{attribute 'linkalways'} 
{attribute 'no_explicit_call' := 'This FB is a CLASS and must be accessed using methods or properties'}
{attribute 'enable_dynamic_creation'}
FUNCTION_BLOCK Node_F_VN_ConvertCartesianToPolarPoints EXTENDS VisionNode
VAR
	ipSrcPointsCart : _ITcVnContainer;
    ipDestPointsPolar : _ITcVnContainer;
    hrPrev : _HRESULT(S_OK);
	hresult : _HRESULT(S_OK);
END_VAR

METHOD PUBLIC  Clone : I_Node
VAR
	pNode : POINTER TO Node_F_VN_ConvertCartesianToPolarPoints;
END_VAR
pNode := __NEW(Node_F_VN_ConvertCartesianToPolarPoints);
Clone := pNode^;
END_METHOD

METHOD FB_init : BOOL
VAR_INPUT
	bInitRetains : BOOL; // if TRUE, the retain variables are initialized (warm start / cold start)
	bInCopyCode : BOOL;  // if TRUE, the instance afterwards gets moved into the copy code (online change)
END_VAR
AddInput('ipSrcPointsCart', ipSrcPointsCart);
AddInput('hrPrev', hrPrev);
AddOutput('ipDestPointsPolar', ipDestPointsPolar);
AddOutput('hresult',hresult);
END_METHOD

METHOD PROTECTED OnExecute
hresult.Value := F_VN_ConvertCartesianToPolarPoints(
	ipSrcPointsCart := ipSrcPointsCart.Value,
	ipDestPointsPolar := ipDestPointsPolar.Value,
	hrPrev := hrPrev.Value);
END_METHOD

METHOD PUBLIC PreExecutionCheck
VAR_INPUT
	Check : I_PreExecutionChecks;
END_VAR
Check.IsTrue(ipSrcPointsCart.IsValid, 'ipSrcPointsCart must be a valid container');
Check.IsTrue((ipSrcPointsCart.IsType(TC_GLOBAL_CONST_LIST.ContainerType_Vector_TcVnPoint2_DINT) OR
              ipSrcPointsCart.IsType(TC_GLOBAL_CONST_LIST.ContainerType_Vector_TcVnPoint2_REAL) OR
              ipSrcPointsCart.IsType(TC_GLOBAL_CONST_LIST.ContainerType_Vector_TcVnPoint2_LREAL)),
              'ipSrcPointsCart contains incorrect type');
END_METHOD

END_FUNCTION_BLOCK

(* stored: Version 1.1.0.1, ProductVersion 3.1.4026.13
   POU Node_F_VN_ConvertCartesianToPolarPoints: Id {aa9d6711-de47-0550-3f79-16dbf31c8122}, SpecialFunc None
   Folder Constructor: Id {8debbfbf-b0de-00a3-16d6-1cacd434fbc6}
   Method Clone: Id {73d90da3-98b5-0e78-13fb-aba62421fb7d}
   Method FB_init: Id {546389e7-6c41-0724-2b32-1f2025db1a58}
   Method OnExecute: Id {01124f60-7a7e-022f-038e-f3bbc39c3b7b}
   Method PreExecutionCheck: Id {e0dc8598-73de-0a27-0ddf-532fabe60ee8} *)
